// TIA Portal V20 export
TYPE "UDT_HMI_SeñalesGalibo"
   STRUCT
      Alt_0_PaletVacio : Bool;
      Alt_1 : Bool;
      Alt_2 : Bool;
      Alt_3 : Bool;
      Alt_4 : Bool;
      Alt_Err : Bool;
      Anch_Der_1 : Bool;
      Anch_Der_2 : Bool;
      Anch_Der_3 : Bool;
      Anch_Der_Err : Bool;
      Anch_Izq_1 : Bool;
      Anch_Izq_2 : Bool;
      Anch_Izq_3 : Bool;
      Anch_Izq_Err : Bool;
      Front_1 : Bool;
      Front_2 : Bool;
      Front_3 : Bool;
      Hueco : Bool;
      HuecoRemon : Bool;
      Patin_1 : Bool;
      Patin_2 : Bool;
      Baliza : Bool;
      Frontal_Del_1 : Bool;
      Frontal_Del_2 : Bool;
      Frontal_Del_Err : Bool;
      Frontal_Tra_1 : Bool;
      Frontal_Tra_2 : Bool;
      Frontal_Tra_Err : Bool;
      Reserva_1 : Bool;
      Reserva_2 : Bool;
      Reserva_3 : Bool;
      Reserva_4 : Bool;
   END_STRUCT;
END_TYPE
